													(
														ParameterName_as8		:=	'Maschinentyp',
														ParameterType_u8		:= 1,
														attr1_u					:= 1,
														attr2_u					:= 5,
														attr3_u					:= 1,
														UnitCode_au8			:= 0,
														Multiplier_s16			:= 1,
														Divisor_s16				:= 1,
														NumberOfDigits_u16	:= 0,
														AccesslevelCode_u8	:= 3,
														attr4_u					:= 1,
														EEPROMAddress_s		:= (Page_u8 := 3, IntIndex_u8 := 0)
													)

											)

										),

										(
											MenuName_as8 :=	'Menu 1',

											ParameterGroup_as :=

											(
												GroupName_as8	:=	'Maschine',

												Param_as 		:=

													(
														ParameterName_as8		:=	'Maschinentyp',
														ParameterType_u8		:= 1,
														attr1_u					:= 1,
														attr2_u					:= 5,
														attr3_u					:= 1,
														UnitCode_au8			:= 0,
														Multiplier_s16			:= 1,
														Divisor_s16				:= 1,
														NumberOfDigits_u16	:= 0,
														AccesslevelCode_u8	:= 3,
														attr4_u					:= 1,
														EEPROMAddress_s		:= (Page_u8 := 3, IntIndex_u8 := 0)
													),


													(
														ParameterName_as8		:=	'Maschinentyp',
														ParameterType_u8		:= 1,
														attr1_u					:= 1,
														attr2_u					:= 5,
														attr3_u					:= 1,
														UnitCode_au8			:= 0,
														Multiplier_s16			:= 1,
														Divisor_s16				:= 1,
														NumberOfDigits_u16	:= 0,
														AccesslevelCode_u8	:= 3,
														attr4_u					:= 1,
														EEPROMAddress_s		:= (Page_u8 := 3, IntIndex_u8 := 0)
													),



													(
														ParameterName_as8		:=	'Maschinentyp',
														ParameterType_u8		:= 1,
														attr1_u					:= 1,
														attr2_u					:= 5,
														attr3_u					:= 1,
														UnitCode_au8			:= 0,
														Multiplier_s16			:= 1,
														Divisor_s16				:= 1,
														NumberOfDigits_u16	:= 0,
														AccesslevelCode_u8	:= 3,
														attr4_u					:= 1,
														EEPROMAddress_s		:= (Page_u8 := 3, IntIndex_u8 := 0)
													),



													(
														ParameterName_as8		:=	'Maschinentyp',
														ParameterType_u8		:= 1,
														attr1_u					:= 1,
														attr2_u					:= 5,
														attr3_u					:= 1,
														UnitCode_au8			:= 0,
														Multiplier_s16			:= 1,
														Divisor_s16				:= 1,
														NumberOfDigits_u16	:= 0,
														AccesslevelCode_u8	:= 3,
														attr4_u					:= 1,
														EEPROMAddress_s		:= (Page_u8 := 3, IntIndex_u8 := 0)
													),



													(
														ParameterName_as8		:=	'Maschinentyp',
														ParameterType_u8		:= 1,
														attr1_u					:= 1,
														attr2_u					:= 5,
														attr3_u					:= 1,
														UnitCode_au8			:= 0,
														Multiplier_s16			:= 1,
														Divisor_s16				:= 1,
														NumberOfDigits_u16	:= 0,
														AccesslevelCode_u8	:= 3,
														attr4_u					:= 1,
														EEPROMAddress_s		:= (Page_u8 := 3, IntIndex_u8 := 0)
													),


													(
														ParameterName_as8		:=	'Maschinentyp',
														ParameterType_u8		:= 1,
														attr1_u					:= 1,
														attr2_u					:= 5,
														attr3_u					:= 1,
														UnitCode_au8			:= 0,
														Multiplier_s16			:= 1,
														Divisor_s16				:= 1,
														NumberOfDigits_u16	:= 0,
														AccesslevelCode_u8	:= 3,
														attr4_u					:= 1,
														EEPROMAddress_s		:= (Page_u8 := 3, IntIndex_u8 := 0)
													),



													(
														ParameterName_as8		:=	'Maschinentyp',
														ParameterType_u8		:= 1,
														attr1_u					:= 1,
														attr2_u					:= 5,
														attr3_u					:= 1,
														UnitCode_au8			:= 0,
														Multiplier_s16			:= 1,
														Divisor_s16				:= 1,
														NumberOfDigits_u16	:= 0,
														AccesslevelCode_u8	:= 3,
														attr4_u					:= 1,
														EEPROMAddress_s		:= (Page_u8 := 3, IntIndex_u8 := 0)
													),


													(
														ParameterName_as8		:=	'Maschinentyp',
														ParameterType_u8		:= 1,
														attr1_u					:= 1,
														attr2_u					:= 5,
														attr3_u					:= 1,
														UnitCode_au8			:= 0,
														Multiplier_s16			:= 1,
														Divisor_s16				:= 1,
														NumberOfDigits_u16	:= 0,
														AccesslevelCode_u8	:= 3,
														attr4_u					:= 1,
														EEPROMAddress_s		:= (Page_u8 := 3, IntIndex_u8 := 0)
													)

											),


											(
												GroupName_as8	:=	'Maschine',

												Param_as 		:=

													(
														ParameterName_as8		:=	'Maschinentyp',
														ParameterType_u8		:= 1,
														attr1_u					:= 1,
														attr2_u					:= 5,
														attr3_u					:= 1,
														UnitCode_au8			:= 0,
														Multiplier_s16			:= 1,
														Divisor_s16				:= 1,
														NumberOfDigits_u16	:= 0,
														AccesslevelCode_u8	:= 3,
														attr4_u					:= 1,
														EEPROMAddress_s		:= (Page_u8 := 3, IntIndex_u8 := 0)
													),


													(
														ParameterName_as8		:=	'Maschinentyp',
														ParameterType_u8		:= 1,
														attr1_u					:= 1,
														attr2_u					:= 5,
														attr3_u					:= 1,
														UnitCode_au8			:= 0,
														Multiplier_s16			:= 1,
														Divisor_s16				:= 1,
														NumberOfDigits_u16	:= 0,
														AccesslevelCode_u8	:= 3,
														attr4_u					:= 1,
														EEPROMAddress_s		:= (Page_u8 := 3, IntIndex_u8 := 0)
													),



													(
														ParameterName_as8		:=	'Maschinentyp',
														ParameterType_u8		:= 1,
														attr1_u					:= 1,
														attr2_u					:= 5,
														attr3_u					:= 1,
														UnitCode_au8			:= 0,
														Multiplier_s16			:= 1,
														Divisor_s16				:= 1,
														NumberOfDigits_u16	:= 0,
														AccesslevelCode_u8	:= 3,
														attr4_u					:= 1,
														EEPROMAddress_s		:= (Page_u8 := 3, IntIndex_u8 := 0)
													),



													(
														ParameterName_as8		:=	'Maschinentyp',
														ParameterType_u8		:= 1,
														attr1_u					:= 1,
														attr2_u					:= 5,
														attr3_u					:= 1,
														UnitCode_au8			:= 0,
														Multiplier_s16			:= 1,
														Divisor_s16				:= 1,
														NumberOfDigits_u16	:= 0,
														AccesslevelCode_u8	:= 3,
														attr4_u					:= 1,
														EEPROMAddress_s		:= (Page_u8 := 3, IntIndex_u8 := 0)
													),



													(
														ParameterName_as8		:=	'Maschinentyp',
														ParameterType_u8		:= 1,
														attr1_u					:= 1,
														attr2_u					:= 5,
														attr3_u					:= 1,
														UnitCode_au8			:= 0,
														Multiplier_s16			:= 1,
														Divisor_s16				:= 1,
														NumberOfDigits_u16	:= 0,
														AccesslevelCode_u8	:= 3,
														attr4_u					:= 1,
														EEPROMAddress_s		:= (Page_u8 := 3, IntIndex_u8 := 0)
													),


													(
														ParameterName_as8		:=	'Maschinentyp',
														ParameterType_u8		:= 1,
														attr1_u					:= 1,
														attr2_u					:= 5,
														attr3_u					:= 1,
														UnitCode_au8			:= 0,
														Multiplier_s16			:= 1,
														Divisor_s16				:= 1,
														NumberOfDigits_u16	:= 0,
														AccesslevelCode_u8	:= 3,
														attr4_u					:= 1,
														EEPROMAddress_s		:= (Page_u8 := 3, IntIndex_u8 := 0)
													),



													(
														ParameterName_as8		:=	'Maschinentyp',
														ParameterType_u8		:= 1,
														attr1_u					:= 1,
														attr2_u					:= 5,
														attr3_u					:= 1,
														UnitCode_au8			:= 0,
														Multiplier_s16			:= 1,
														Divisor_s16				:= 1,
														NumberOfDigits_u16	:= 0,
														AccesslevelCode_u8	:= 3,
														attr4_u					:= 1,
														EEPROMAddress_s		:= (Page_u8 := 3, IntIndex_u8 := 0)
													),


													(
														ParameterName_as8		:=	'Maschinentyp',
														ParameterType_u8		:= 1,
														attr1_u					:= 1,
														attr2_u					:= 5,
														attr3_u					:= 1,
														UnitCode_au8			:= 0,
														Multiplier_s16			:= 1,
														Divisor_s16				:= 1,
														NumberOfDigits_u16	:= 0,
														AccesslevelCode_u8	:= 3,
														attr4_u					:= 1,
														EEPROMAddress_s		:= (Page_u8 := 3, IntIndex_u8 := 0)
													)

											),


											(
												GroupName_as8	:=	'Maschine',

												Param_as 		:=

													(
														ParameterName_as8		:=	'Maschinentyp',
														ParameterType_u8		:= 1,
														attr1_u					:= 1,
														attr2_u					:= 5,
														attr3_u					:= 1,
														UnitCode_au8			:= 0,
														Multiplier_s16			:= 1,
														Divisor_s16				:= 1,
														NumberOfDigits_u16	:= 0,
														AccesslevelCode_u8	:= 3,
														attr4_u					:= 1,
														EEPROMAddress_s		:= (Page_u8 := 3, IntIndex_u8 := 0)
													),


													(
														ParameterName_as8		:=	'Maschinentyp',
														ParameterType_u8		:= 1,
														attr1_u					:= 1,
														attr2_u					:= 5,
														attr3_u					:= 1,
														UnitCode_au8			:= 0,
														Multiplier_s16			:= 1,
														Divisor_s16				:= 1,
														NumberOfDigits_u16	:= 0,
														AccesslevelCode_u8	:= 3,
														attr4_u					:= 1,
														EEPROMAddress_s		:= (Page_u8 := 3, IntIndex_u8 := 0)
													),



													(
														ParameterName_as8		:=	'Maschinentyp',
														ParameterType_u8		:= 1,
														attr1_u					:= 1,
														attr2_u					:= 5,
														attr3_u					:= 1,
														UnitCode_au8			:= 0,
														Multiplier_s16			:= 1,
														Divisor_s16				:= 1,
														NumberOfDigits_u16	:= 0,
														AccesslevelCode_u8	:= 3,
														attr4_u					:= 1,
														EEPROMAddress_s		:= (Page_u8 := 3, IntIndex_u8 := 0)
													),



													(
														ParameterName_as8		:=	'Maschinentyp',
														ParameterType_u8		:= 1,
														attr1_u					:= 1,
														attr2_u					:= 5,
														attr3_u					:= 1,
														UnitCode_au8			:= 0,
														Multiplier_s16			:= 1,
														Divisor_s16				:= 1,
														NumberOfDigits_u16	:= 0,
														AccesslevelCode_u8	:= 3,
														attr4_u					:= 1,
														EEPROMAddress_s		:= (Page_u8 := 3, IntIndex_u8 := 0)
													),



													(
														ParameterName_as8		:=	'Maschinentyp',
														ParameterType_u8		:= 1,
														attr1_u					:= 1,
														attr2_u					:= 5,
														attr3_u					:= 1,
														UnitCode_au8			:= 0,
														Multiplier_s16			:= 1,
														Divisor_s16				:= 1,
														NumberOfDigits_u16	:= 0,
														AccesslevelCode_u8	:= 3,
														attr4_u					:= 1,
														EEPROMAddress_s		:= (Page_u8 := 3, IntIndex_u8 := 0)
													),


													(
														ParameterName_as8		:=	'Maschinentyp',
														ParameterType_u8		:= 1,
														attr1_u					:= 1,
														attr2_u					:= 5,
														attr3_u					:= 1,
														UnitCode_au8			:= 0,
														Multiplier_s16			:= 1,
														Divisor_s16				:= 1,
														NumberOfDigits_u16	:= 0,
														AccesslevelCode_u8	:= 3,
														attr4_u					:= 1,
														EEPROMAddress_s		:= (Page_u8 := 3, IntIndex_u8 := 0)
													),



													(
														ParameterName_as8		:=	'Maschinentyp',
														ParameterType_u8		:= 1,
														attr1_u					:= 1,
														attr2_u					:= 5,
														attr3_u					:= 1,
														UnitCode_au8			:= 0,
														Multiplier_s16			:= 1,
														Divisor_s16				:= 1,
														NumberOfDigits_u16	:= 0,
														AccesslevelCode_u8	:= 3,
														attr4_u					:= 1,
														EEPROMAddress_s		:= (Page_u8 := 3, IntIndex_u8 := 0)
													),


													(
														ParameterName_as8		:=	'Maschinentyp',
														ParameterType_u8		:= 1,
														attr1_u					:= 1,
														attr2_u					:= 5,
														attr3_u					:= 1,
														UnitCode_au8			:= 0,
														Multiplier_s16			:= 1,
														Divisor_s16				:= 1,
														NumberOfDigits_u16	:= 0,
														AccesslevelCode_u8	:= 3,
														attr4_u					:= 1,
														EEPROMAddress_s		:= (Page_u8 := 3, IntIndex_u8 := 0)
													)

											),


											(
												GroupName_as8	:=	'Maschine',

												Param_as 		:=

													(
														ParameterName_as8		:=	'Maschinentyp',
														ParameterType_u8		:= 1,
														attr1_u					:= 1,
														attr2_u					:= 5,
														attr3_u					:= 1,
														UnitCode_au8			:= 0,
														Multiplier_s16			:= 1,
														Divisor_s16				:= 1,
														NumberOfDigits_u16	:= 0,
														AccesslevelCode_u8	:= 3,
														attr4_u					:= 1,
														EEPROMAddress_s		:= (Page_u8 := 3, IntIndex_u8 := 0)
													),


													(
														ParameterName_as8		:=	'Maschinentyp',
														ParameterType_u8		:= 1,
														attr1_u					:= 1,
														attr2_u					:= 5,
														attr3_u					:= 1,
														UnitCode_au8			:= 0,
														Multiplier_s16			:= 1,
														Divisor_s16				:= 1,
														NumberOfDigits_u16	:= 0,
														AccesslevelCode_u8	:= 3,
														attr4_u					:= 1,
														EEPROMAddress_s		:= (Page_u8 := 3, IntIndex_u8 := 0)
													),



													(
														ParameterName_as8		:=	'Maschinentyp',
														ParameterType_u8		:= 1,
														attr1_u					:= 1,
														attr2_u					:= 5,
														attr3_u					:= 1,
														UnitCode_au8			:= 0,
														Multiplier_s16			:= 1,
														Divisor_s16				:= 1,
														NumberOfDigits_u16	:= 0,
														AccesslevelCode_u8	:= 3,
														attr4_u					:= 1,
														EEPROMAddress_s		:= (Page_u8 := 3, IntIndex_u8 := 0)
													),



													(
														ParameterName_as8		:=	'Maschinentyp',
														ParameterType_u8		:= 1,
														attr1_u					:= 1,
														attr2_u					:= 5,
														attr3_u					:= 1,
														UnitCode_au8			:= 0,
														Multiplier_s16			:= 1,
														Divisor_s16				:= 1,
														NumberOfDigits_u16	:= 0,
														AccesslevelCode_u8	:= 3,
														attr4_u					:= 1,
														EEPROMAddress_s		:= (Page_u8 := 3, IntIndex_u8 := 0)
													),



													(
														ParameterName_as8		:=	'Maschinentyp',
														ParameterType_u8		:= 1,
														attr1_u					:= 1,
														attr2_u					:= 5,
														attr3_u					:= 1,
														UnitCode_au8			:= 0,
														Multiplier_s16			:= 1,
														Divisor_s16				:= 1,
														NumberOfDigits_u16	:= 0,
														AccesslevelCode_u8	:= 3,
														attr4_u					:= 1,
														EEPROMAddress_s		:= (Page_u8 := 3, IntIndex_u8 := 0)
													),


													(
														ParameterName_as8		:=	'Maschinentyp',
														ParameterType_u8		:= 1,
														attr1_u					:= 1,
														attr2_u					:= 5,
														attr3_u					:= 1,
														UnitCode_au8			:= 0,
														Multiplier_s16			:= 1,
														Divisor_s16				:= 1,
														NumberOfDigits_u16	:= 0,
														AccesslevelCode_u8	:= 3,
														attr4_u					:= 1,
														EEPROMAddress_s		:= (Page_u8 := 3, IntIndex_u8 := 0)
													),



													(
														ParameterName_as8		:=	'Maschinentyp',
														ParameterType_u8		:= 1,
														attr1_u					:= 1,
														attr2_u					:= 5,
														attr3_u					:= 1,
														UnitCode_au8			:= 0,
														Multiplier_s16			:= 1,
														Divisor_s16				:= 1,
														NumberOfDigits_u16	:= 0,
														AccesslevelCode_u8	:= 3,
														attr4_u					:= 1,
														EEPROMAddress_s		:= (Page_u8 := 3, IntIndex_u8 := 0)
													),


													(
														ParameterName_as8		:=	'Maschinentyp',
														ParameterType_u8		:= 1,
														attr1_u					:= 1,
														attr2_u					:= 5,
														attr3_u					:= 1,
														UnitCode_au8			:= 0,
														Multiplier_s16			:= 1,
														Divisor_s16				:= 1,
														NumberOfDigits_u16	:= 0,
														AccesslevelCode_u8	:= 3,
														attr4_u					:= 1,
														EEPROMAddress_s		:= (Page_u8 := 3, IntIndex_u8 := 0)
													)

											),


											(
												GroupName_as8	:=	'Maschine',

												Param_as 		:=

													(
														ParameterName_as8		:=	'Maschinentyp',
														ParameterType_u8		:= 1,
														attr1_u					:= 1,
														attr2_u					:= 5,
														attr3_u					:= 1,
														UnitCode_au8			:= 0,
														Multiplier_s16			:= 1,
														Divisor_s16				:= 1,
														NumberOfDigits_u16	:= 0,
														AccesslevelCode_u8	:= 3,
														attr4_u					:= 1,
														EEPROMAddress_s		:= (Page_u8 := 3, IntIndex_u8 := 0)
													),


													(
														ParameterName_as8		:=	'Maschinentyp',
														ParameterType_u8		:= 1,
														attr1_u					:= 1,
														attr2_u					:= 5,
														attr3_u					:= 1,
														UnitCode_au8			:= 0,
														Multiplier_s16			:= 1,
														Divisor_s16				:= 1,
														NumberOfDigits_u16	:= 0,
														AccesslevelCode_u8	:= 3,
														attr4_u					:= 1,
														EEPROMAddress_s		:= (Page_u8 := 3, IntIndex_u8 := 0)
													),



													(
														ParameterName_as8		:=	'Maschinentyp',
														ParameterType_u8		:= 1,
														attr1_u					:= 1,
														attr2_u					:= 5,
														attr3_u					:= 1,
														UnitCode_au8			:= 0,
														Multiplier_s16			:= 1,
														Divisor_s16				:= 1,
														NumberOfDigits_u16	:= 0,
														AccesslevelCode_u8	:= 3,
														attr4_u					:= 1,
														EEPROMAddress_s		:= (Page_u8 := 3, IntIndex_u8 := 0)
													),



													(
														ParameterName_as8		:=	'Maschinentyp',
														ParameterType_u8		:= 1,
														attr1_u					:= 1,
														attr2_u					:= 5,
														attr3_u					:= 1,
														UnitCode_au8			:= 0,
														Multiplier_s16			:= 1,
														Divisor_s16				:= 1,
														NumberOfDigits_u16	:= 0,
														AccesslevelCode_u8	:= 3,
														attr4_u					:= 1,
														EEPROMAddress_s		:= (Page_u8 := 3, IntIndex_u8 := 0)
													),



													(
														ParameterName_as8		:=	'Maschinentyp',
														ParameterType_u8		:= 1,
														attr1_u					:= 1,
														attr2_u					:= 5,
														attr3_u					:= 1,
														UnitCode_au8			:= 0,
														Multiplier_s16			:= 1,
														Divisor_s16				:= 1,
														NumberOfDigits_u16	:= 0,
														AccesslevelCode_u8	:= 3,
														attr4_u					:= 1,
														EEPROMAddress_s		:= (Page_u8 := 3, IntIndex_u8 := 0)
													),


													(
														ParameterName_as8		:=	'Maschinentyp',
														ParameterType_u8		:= 1,
														attr1_u					:= 1,
														attr2_u					:= 5,
														attr3_u					:= 1,
														UnitCode_au8			:= 0,
														Multiplier_s16			:= 1,
														Divisor_s16				:= 1,
														NumberOfDigits_u16	:= 0,
														AccesslevelCode_u8	:= 3,
														attr4_u					:= 1,
														EEPROMAddress_s		:= (Page_u8 := 3, IntIndex_u8 := 0)
													),



													(
														ParameterName_as8		:=	'Maschinentyp',
														ParameterType_u8		:= 1,
														attr1_u					:= 1,
														attr2_u					:= 5,
														attr3_u					:= 1,
														UnitCode_au8			:= 0,
														Multiplier_s16			:= 1,
														Divisor_s16				:= 1,
														NumberOfDigits_u16	:= 0,
														AccesslevelCode_u8	:= 3,
														attr4_u					:= 1,
														EEPROMAddress_s		:= (Page_u8 := 3, IntIndex_u8 := 0)
													),


													(
														ParameterName_as8		:=	'Maschinentyp',
														ParameterType_u8		:= 1,
														attr1_u					:= 1,
														attr2_u					:= 5,
														attr3_u					:= 1,
														UnitCode_au8			:= 0,
														Multiplier_s16			:= 1,
														Divisor_s16				:= 1,
														NumberOfDigits_u16	:= 0,
														AccesslevelCode_u8	:= 3,
														attr4_u					:= 1,
														EEPROMAddress_s		:= (Page_u8 := 3, IntIndex_u8 := 0)
													)

											),


											(
												GroupName_as8	:=	'Maschine',

												Param_as 		:=

													(
														ParameterName_as8		:=	'Maschinentyp',
														ParameterType_u8		:= 1,
														attr1_u					:= 1,
														attr2_u					:= 5,
														attr3_u					:= 1,
														UnitCode_au8			:= 0,
														Multiplier_s16			:= 1,
														Divisor_s16				:= 1,
														NumberOfDigits_u16	:= 0,
														AccesslevelCode_u8	:= 3,
														attr4_u					:= 1,
														EEPROMAddress_s		:= (Page_u8 := 3, IntIndex_u8 := 0)
													),


													(
														ParameterName_as8		:=	'Maschinentyp',
														ParameterType_u8		:= 1,
														attr1_u					:= 1,
														attr2_u					:= 5,
														attr3_u					:= 1,
														UnitCode_au8			:= 0,
														Multiplier_s16			:= 1,
														Divisor_s16				:= 1,
														NumberOfDigits_u16	:= 0,
														AccesslevelCode_u8	:= 3,
														attr4_u					:= 1,
														EEPROMAddress_s		:= (Page_u8 := 3, IntIndex_u8 := 0)
													),



													(
														ParameterName_as8		:=	'Maschinentyp',
														ParameterType_u8		:= 1,
														attr1_u					:= 1,
														attr2_u					:= 5,
														attr3_u					:= 1,
														UnitCode_au8			:= 0,
														Multiplier_s16			:= 1,
														Divisor_s16				:= 1,
														NumberOfDigits_u16	:= 0,
														AccesslevelCode_u8	:= 3,
														attr4_u					:= 1,
														EEPROMAddress_s		:= (Page_u8 := 3, IntIndex_u8 := 0)
													),



													(
														ParameterName_as8		:=	'Maschinentyp',
														ParameterType_u8		:= 1,
														attr1_u					:= 1,
														attr2_u					:= 5,
														attr3_u					:= 1,
														UnitCode_au8			:= 0,
														Multiplier_s16			:= 1,
														Divisor_s16				:= 1,
														NumberOfDigits_u16	:= 0,
														AccesslevelCode_u8	:= 3,
														attr4_u					:= 1,
														EEPROMAddress_s		:= (Page_u8 := 3, IntIndex_u8 := 0)
													),



													(
														ParameterName_as8		:=	'Maschinentyp',
														ParameterType_u8		:= 1,
														attr1_u					:= 1,
														attr2_u					:= 5,
														attr3_u					:= 1,
														UnitCode_au8			:= 0,
														Multiplier_s16			:= 1,
														Divisor_s16				:= 1,
														NumberOfDigits_u16	:= 0,
														AccesslevelCode_u8	:= 3,
														attr4_u					:= 1,
														EEPROMAddress_s		:= (Page_u8 := 3, IntIndex_u8 := 0)
													),


													(
														ParameterName_as8		:=	'Maschinentyp',
														ParameterType_u8		:= 1,
														attr1_u					:= 1,
														attr2_u					:= 5,
														attr3_u					:= 1,
														UnitCode_au8			:= 0,
														Multiplier_s16			:= 1,
														Divisor_s16				:= 1,
														NumberOfDigits_u16	:= 0,
														AccesslevelCode_u8	:= 3,
														attr4_u					:= 1,
														EEPROMAddress_s		:= (Page_u8 := 3, IntIndex_u8 := 0)
													),



													(
														ParameterName_as8		:=	'Maschinentyp',
														ParameterType_u8		:= 1,
														attr1_u					:= 1,
														attr2_u					:= 5,
														attr3_u					:= 1,
														UnitCode_au8			:= 0,
														Multiplier_s16			:= 1,
														Divisor_s16				:= 1,
														NumberOfDigits_u16	:= 0,
														AccesslevelCode_u8	:= 3,
														attr4_u					:= 1,
														EEPROMAddress_s		:= (Page_u8 := 3, IntIndex_u8 := 0)
													),


													(
														ParameterName_as8		:=	'Maschinentyp',
														ParameterType_u8		:= 1,
														attr1_u					:= 1,
														attr2_u					:= 5,
														attr3_u					:= 1,
														UnitCode_au8			:= 0,
														Multiplier_s16			:= 1,
														Divisor_s16				:= 1,
														NumberOfDigits_u16	:= 0,
														AccesslevelCode_u8	:= 3,
														attr4_u					:= 1,
														EEPROMAddress_s		:= (Page_u8 := 3, IntIndex_u8 := 0)
													)

											),


											(
												GroupName_as8	:=	'Maschine',

												Param_as 		:=

													(
														ParameterName_as8		:=	'Maschinentyp',
														ParameterType_u8		:= 1,
														attr1_u					:= 1,
														attr2_u					:= 5,
														attr3_u					:= 1,
														UnitCode_au8			:= 0,
														Multiplier_s16			:= 1,
														Divisor_s16				:= 1,
														NumberOfDigits_u16	:= 0,
														AccesslevelCode_u8	:= 3,
														attr4_u					:= 1,
														EEPROMAddress_s		:= (Page_u8 := 3, IntIndex_u8 := 0)
													),


													(
														ParameterName_as8		:=	'Maschinentyp',
														ParameterType_u8		:= 1,
														attr1_u					:= 1,
														attr2_u					:= 5,
														attr3_u					:= 1,
														UnitCode_au8			:= 0,
														Multiplier_s16			:= 1,
														Divisor_s16				:= 1,
														NumberOfDigits_u16	:= 0,
														AccesslevelCode_u8	:= 3,
														attr4_u					:= 1,
														EEPROMAddress_s		:= (Page_u8 := 3, IntIndex_u8 := 0)
													),



													(
														ParameterName_as8		:=	'Maschinentyp',
														ParameterType_u8		:= 1,
														attr1_u					:= 1,
														attr2_u					:= 5,
														attr3_u					:= 1,
														UnitCode_au8			:= 0,
														Multiplier_s16			:= 1,
														Divisor_s16				:= 1,
														NumberOfDigits_u16	:= 0,
														AccesslevelCode_u8	:= 3,
														attr4_u					:= 1,
														EEPROMAddress_s		:= (Page_u8 := 3, IntIndex_u8 := 0)
													),



													(
														ParameterName_as8		:=	'Maschinentyp',
														ParameterType_u8		:= 1,
														attr1_u					:= 1,
														attr2_u					:= 5,
														attr3_u					:= 1,
														UnitCode_au8			:= 0,
														Multiplier_s16			:= 1,
														Divisor_s16				:= 1,
														NumberOfDigits_u16	:= 0,
														AccesslevelCode_u8	:= 3,
														attr4_u					:= 1,
														EEPROMAddress_s		:= (Page_u8 := 3, IntIndex_u8 := 0)
													),



													(
														ParameterName_as8		:=	'Maschinentyp',
														ParameterType_u8		:= 1,
														attr1_u					:= 1,
														attr2_u					:= 5,
														attr3_u					:= 1,
														UnitCode_au8			:= 0,
														Multiplier_s16			:= 1,
														Divisor_s16				:= 1,
														NumberOfDigits_u16	:= 0,
														AccesslevelCode_u8	:= 3,
														attr4_u					:= 1,
														EEPROMAddress_s		:= (Page_u8 := 3, IntIndex_u8 := 0)
													),


													(
														ParameterName_as8		:=	'Maschinentyp',
														ParameterType_u8		:= 1,
														attr1_u					:= 1,
														attr2_u					:= 5,
														attr3_u					:= 1,
														UnitCode_au8			:= 0,
														Multiplier_s16			:= 1,
														Divisor_s16				:= 1,
														NumberOfDigits_u16	:= 0,
														AccesslevelCode_u8	:= 3,
														attr4_u					:= 1,
														EEPROMAddress_s		:= (Page_u8 := 3, IntIndex_u8 := 0)
													),



													(
														ParameterName_as8		:=	'Maschinentyp',
														ParameterType_u8		:= 1,
														attr1_u					:= 1,
														attr2_u					:= 5,
														attr3_u					:= 1,
														UnitCode_au8			:= 0,
														Multiplier_s16			:= 1,
														Divisor_s16				:= 1,
														NumberOfDigits_u16	:= 0,
														AccesslevelCode_u8	:= 3,
														attr4_u					:= 1,
														EEPROMAddress_s		:= (Page_u8 := 3, IntIndex_u8 := 0)
													),


													(
														ParameterName_as8		:=	'Maschinentyp',
														ParameterType_u8		:= 1,
														attr1_u					:= 1,
														attr2_u					:= 5,
														attr3_u					:= 1,
														UnitCode_au8			:= 0,
														Multiplier_s16			:= 1,
														Divisor_s16				:= 1,
														NumberOfDigits_u16	:= 0,
														AccesslevelCode_u8	:= 3,
														attr4_u					:= 1,
														EEPROMAddress_s		:= (Page_u8 := 3, IntIndex_u8 := 0)
													)

											),


											(
												GroupName_as8	:=	'Maschine',

												Param_as 		:=

													(
														ParameterName_as8		:=	'Maschinentyp',
														ParameterType_u8		:= 1,
														attr1_u					:= 1,
														attr2_u					:= 5,
														attr3_u					:= 1,
														UnitCode_au8			:= 0,
														Multiplier_s16			:= 1,
														Divisor_s16				:= 1,
														NumberOfDigits_u16	:= 0,
														AccesslevelCode_u8	:= 3,
														attr4_u					:= 1,
														EEPROMAddress_s		:= (Page_u8 := 3, IntIndex_u8 := 0)
													),


													(
														ParameterName_as8		:=	'Maschinentyp',
														ParameterType_u8		:= 1,
														attr1_u					:= 1,
														attr2_u					:= 5,
														attr3_u					:= 1,
														UnitCode_au8			:= 0,
														Multiplier_s16			:= 1,
														Divisor_s16				:= 1,
														NumberOfDigits_u16	:= 0,
														AccesslevelCode_u8	:= 3,
														attr4_u					:= 1,
														EEPROMAddress_s		:= (Page_u8 := 3, IntIndex_u8 := 0)
													),



													(
														ParameterName_as8		:=	'Maschinentyp',
														ParameterType_u8		:= 1,
														attr1_u					:= 1,
														attr2_u					:= 5,
														attr3_u					:= 1,
														UnitCode_au8			:= 0,
														Multiplier_s16			:= 1,
														Divisor_s16				:= 1,
														NumberOfDigits_u16	:= 0,
														AccesslevelCode_u8	:= 3,
														attr4_u					:= 1,
														EEPROMAddress_s		:= (Page_u8 := 3, IntIndex_u8 := 0)
													),



													(
														ParameterName_as8		:=	'Maschinentyp',
														ParameterType_u8		:= 1,
														attr1_u					:= 1,
														attr2_u					:= 5,
														attr3_u					:= 1,
														UnitCode_au8			:= 0,
														Multiplier_s16			:= 1,
														Divisor_s16				:= 1,
														NumberOfDigits_u16	:= 0,
														AccesslevelCode_u8	:= 3,
														attr4_u					:= 1,
														EEPROMAddress_s		:= (Page_u8 := 3, IntIndex_u8 := 0)
													),



													(
														ParameterName_as8		:=	'Maschinentyp',
														ParameterType_u8		:= 1,
														attr1_u					:= 1,
														attr2_u					:= 5,
														attr3_u					:= 1,
														UnitCode_au8			:= 0,
														Multiplier_s16			:= 1,
														Divisor_s16				:= 1,
														NumberOfDigits_u16	:= 0,
														AccesslevelCode_u8	:= 3,
														attr4_u					:= 1,
														EEPROMAddress_s		:= (Page_u8 := 3, IntIndex_u8 := 0)
													),


													(
														ParameterName_as8		:=	'Maschinentyp',
														ParameterType_u8		:= 1,
														attr1_u					:= 1,
														attr2_u					:= 5,
														attr3_u					:= 1,
														UnitCode_au8			:= 0,
														Multiplier_s16			:= 1,
														Divisor_s16				:= 1,
														NumberOfDigits_u16	:= 0,
														AccesslevelCode_u8	:= 3,
														attr4_u					:= 1,
														EEPROMAddress_s		:= (Page_u8 := 3, IntIndex_u8 := 0)
													),



													(
														ParameterName_as8		:=	'Maschinentyp',
														ParameterType_u8		:= 1,
														attr1_u					:= 1,
														attr2_u					:= 5,
														attr3_u					:= 1,
														UnitCode_au8			:= 0,
														Multiplier_s16			:= 1,
														Divisor_s16				:= 1,
														NumberOfDigits_u16	:= 0,
														AccesslevelCode_u8	:= 3,
														attr4_u					:= 1,
														EEPROMAddress_s		:= (Page_u8 := 3, IntIndex_u8 := 0)
													),


													(
														ParameterName_as8		:=	'Maschinentyp',
														ParameterType_u8		:= 1,
														attr1_u					:= 1,
														attr2_u					:= 5,
														attr3_u					:= 1,
														UnitCode_au8			:= 0,
														Multiplier_s16			:= 1,
														Divisor_s16				:= 1,
														NumberOfDigits_u16	:= 0,
														AccesslevelCode_u8	:= 3,
														attr4_u					:= 1,
														EEPROMAddress_s		:= (Page_u8 := 3, IntIndex_u8 := 0)
													)

											)

										);
*)
END_PROGRAM
